KUKA KRL program: art_air.src, art_air.dat

--- art_air.src ---
&ACCESS RV2
DEF art_air ( )

END
; Init air.
GLOBAL DEF ART_air_init ( )
   low_air_signal_timer = 0
END
;
; Air SPS
;
GLOBAL DEF ART_air_SPS()
   IF (NOT isAirPressureOKSignal) THEN
      IF low_air_signal_timer <= 0 THEN
         low_air_signal_timer = ARTTimerGetTime()
      ENDIF

      IF ARTTimerIsTimePassed(low_air_signal_timer, AIR_SIGNAL_OUT_TIME) THEN
         ART_Air_low_preassure = TRUE
      ENDIF
   ELSE
      ART_Air_low_preassure = FALSE
      low_air_signal_timer = 0
   ENDIF
END

--- art_air.dat ---
&ACCESS RV2
DEFDAT  art_air PUBLIC
DECL INT low_air_signal_timer=0
DECL INT AIR_SIGNAL_OUT_TIME=2000
DECL GLOBAL BOOL ART_Air_low_preassure=FALSE
ENDDAT
